SUBAPPLICATION Ventilsteuerung_Uebung_004b3 (* Toggle Flip-Flop mit IE / Split / Verriegelt *)
  (* Standard: 61499-2 *)
  (* Version 1.0, 2023-10-23, franz *)
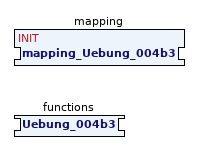
  SUBAPPS
    mapping : mapping_Uebung_004b3;
    functions : Uebung_004b3;
  END_SUBAPPS
END_SUBAPPLICATION
